Staubli VAL3: safety.pgx

program safety()
begin
  while true

    if isPowered()==false

      if esStatus()==0

        put("remise sous pusisance")

        enablePower()

      endIf


    endIf
  endWhile
end
